(* Logix 5000 project; controller TBEN_Lx_8IOL_AOI_V0_2 vendor 1 type 14 code 176 rev 32.11; software revision 32.00; part 14 of 16 *)
(* tags used below, declared in another part *)
   TBEN_I_DATA : INT[173];   // Input Data from IO Block
   TBEN_O_DATA : INT[131];   // Output Data to IO Block
   TBEN_C_DATA : SINT[160];
   DXP1_OUT : BOOL;
   DXP3_OUT : BOOL;
   DXP5_OUT : BOOL;
   DXP7_OUT : BOOL;
   IOLDevice_PORT1 : BOOL;
   IOLDevice_PORT2 : BOOL;
   IOLDevice_PORT3 : BOOL;
   IOLDevice_PORT4 : BOOL;
   IOLDevice_PORT5 : BOOL;
   IOLDevice_PORT6 : BOOL;
   IOLDevice_PORT7 : BOOL;
   IOLDevice_PORT8 : BOOL;
   IOL0_DI : BOOL;
   DXP1_IN : BOOL;
   IOL2_DI : BOOL;
   DXP3_IN : BOOL;
   IOL4_DI : BOOL;
   DXP5_IN : BOOL;
   IOL6_DI : BOOL;
   DXP7_IN : BOOL;
   IOL8_DI : BOOL;
   IOL10_DI : BOOL;
   IOL12_DI : BOOL;
   IOL14_DI : BOOL;
   PORT1_Mode_IOL_or_DI : BOOL;   // 0: IO-LINK without validation 1: Port is set to DI (Power Cycle or Module Inhibit cycle require)
   PORT2_Mode_IOL_or_DI : BOOL;   // 0: IO-LINK without validation 1: Port is set to DI (Power Cycle or Module Inhibit cycle require)
   PORT3_Mode_IOL_or_DI : BOOL;   // 0: IO-LINK without validation 1: Port is set to DI (Power Cycle or Module Inhibit cycle require)
   PORT4_Mode_IOL_or_DI : BOOL;   // 0: IO-LINK without validation 1: Port is set to DI (Power Cycle or Module Inhibit cycle require)
   PORT5_Mode_IOL_or_DI : BOOL;   // 0: IO-LINK without validation 1: Port is set to DI (Power Cycle or Module Inhibit cycle require)
   PORT6_Mode_IOL_or_DI : BOOL;   // 0: IO-LINK without validation 1: Port is set to DI (Power Cycle or Module Inhibit cycle require)
   PORT7_Mode_IOL_or_DI : BOOL;   // 0: IO-LINK without validation 1: Port is set to DI (Power Cycle or Module Inhibit cycle require)
   PORT8_Mode_IOL_or_DI : BOOL;   // 0: IO-LINK without validation 1: Port is set to DI (Power Cycle or Module Inhibit cycle require)
   DisableOutput_DXP1 : BOOL;
   DisableOutput_DXP3 : BOOL;
   DisableOutput_DXP5 : BOOL;
   DisableOutput_DXP7 : BOOL;
   IOLReadActive : BOOL;
   IOLWriteActive : BOOL;
   IOL_READ_Request : BOOL;
   IOL_WRITE_Request : BOOL;
(* TBEN_Lx_8IOL_AOI, continued *)

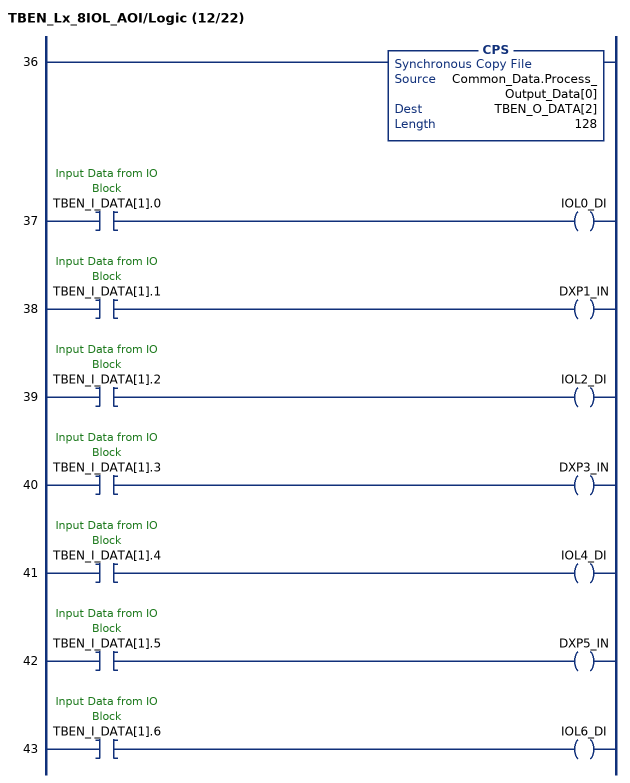
   36: CPS(Common_Data.Process_Output_Data[0],TBEN_O_DATA[2],128);
   37: XIC(TBEN_I_DATA[1].0)OTE(IOL0_DI);
   38: XIC(TBEN_I_DATA[1].1)OTE(DXP1_IN);
   39: XIC(TBEN_I_DATA[1].2)OTE(IOL2_DI);
   40: XIC(TBEN_I_DATA[1].3)OTE(DXP3_IN);
   41: XIC(TBEN_I_DATA[1].4)OTE(IOL4_DI);
   42: XIC(TBEN_I_DATA[1].5)OTE(DXP5_IN);
   43: XIC(TBEN_I_DATA[1].6)OTE(IOL6_DI);
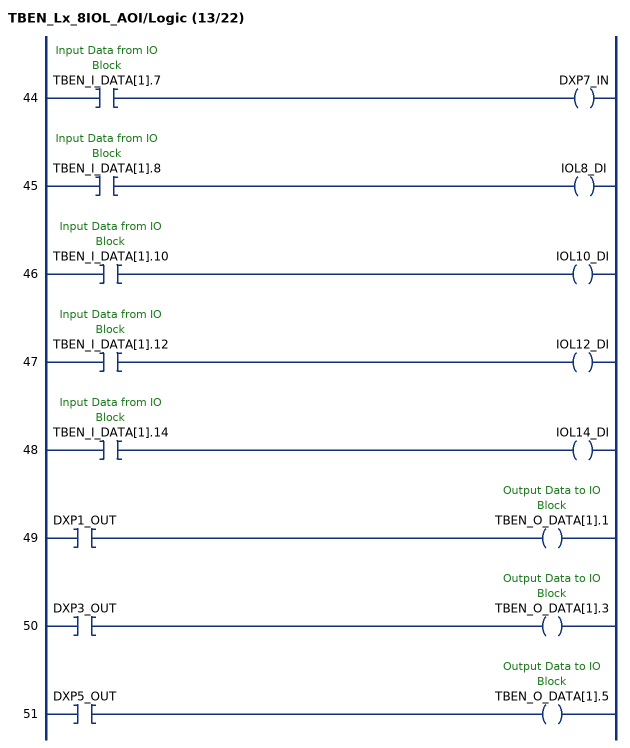
   44: XIC(TBEN_I_DATA[1].7)OTE(DXP7_IN);
   45: XIC(TBEN_I_DATA[1].8)OTE(IOL8_DI);
   46: XIC(TBEN_I_DATA[1].10)OTE(IOL10_DI);
   47: XIC(TBEN_I_DATA[1].12)OTE(IOL12_DI);
   48: XIC(TBEN_I_DATA[1].14)OTE(IOL14_DI);
   49: XIC(DXP1_OUT)OTE(TBEN_O_DATA[1].1);
   50: XIC(DXP3_OUT)OTE(TBEN_O_DATA[1].3);
   51: XIC(DXP5_OUT)OTE(TBEN_O_DATA[1].5);
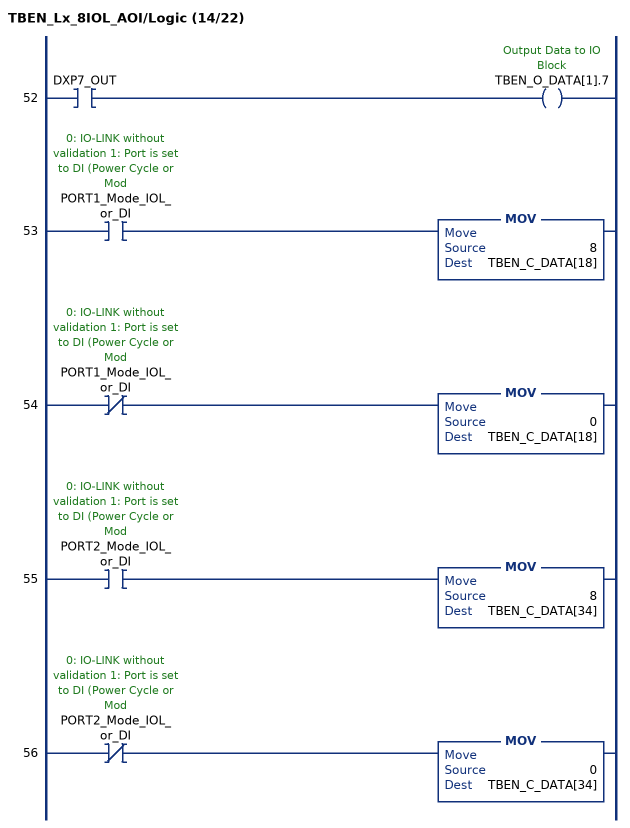
   52: XIC(DXP7_OUT)OTE(TBEN_O_DATA[1].7);
   53: XIC(PORT1_Mode_IOL_or_DI)MOV(8,TBEN_C_DATA[18]);
   54: XIO(PORT1_Mode_IOL_or_DI)MOV(0,TBEN_C_DATA[18]);
   55: XIC(PORT2_Mode_IOL_or_DI)MOV(8,TBEN_C_DATA[34]);
   56: XIO(PORT2_Mode_IOL_or_DI)MOV(0,TBEN_C_DATA[34]);
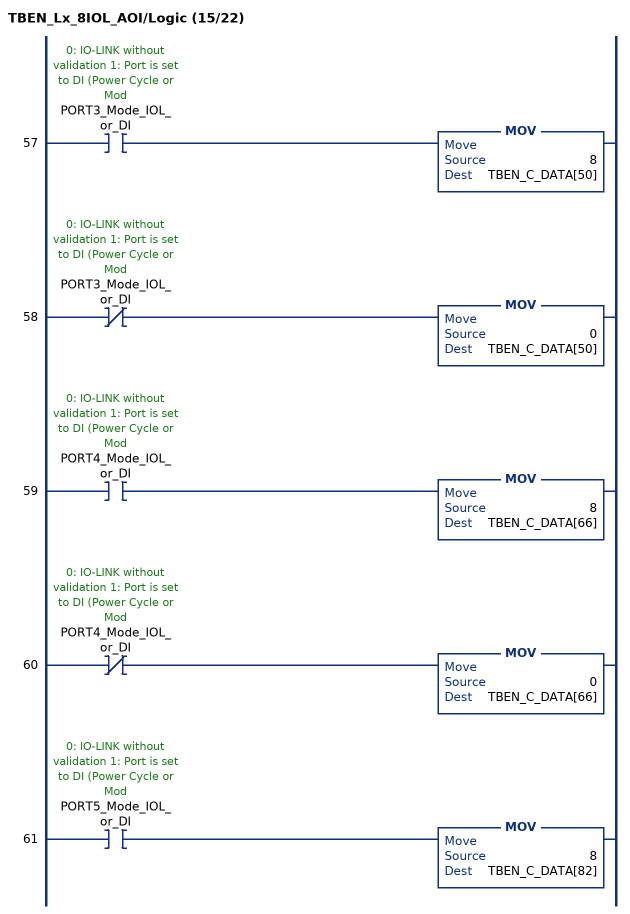
   57: XIC(PORT3_Mode_IOL_or_DI)MOV(8,TBEN_C_DATA[50]);
   58: XIO(PORT3_Mode_IOL_or_DI)MOV(0,TBEN_C_DATA[50]);
   59: XIC(PORT4_Mode_IOL_or_DI)MOV(8,TBEN_C_DATA[66]);
   60: XIO(PORT4_Mode_IOL_or_DI)MOV(0,TBEN_C_DATA[66]);
   61: XIC(PORT5_Mode_IOL_or_DI)MOV(8,TBEN_C_DATA[82]);
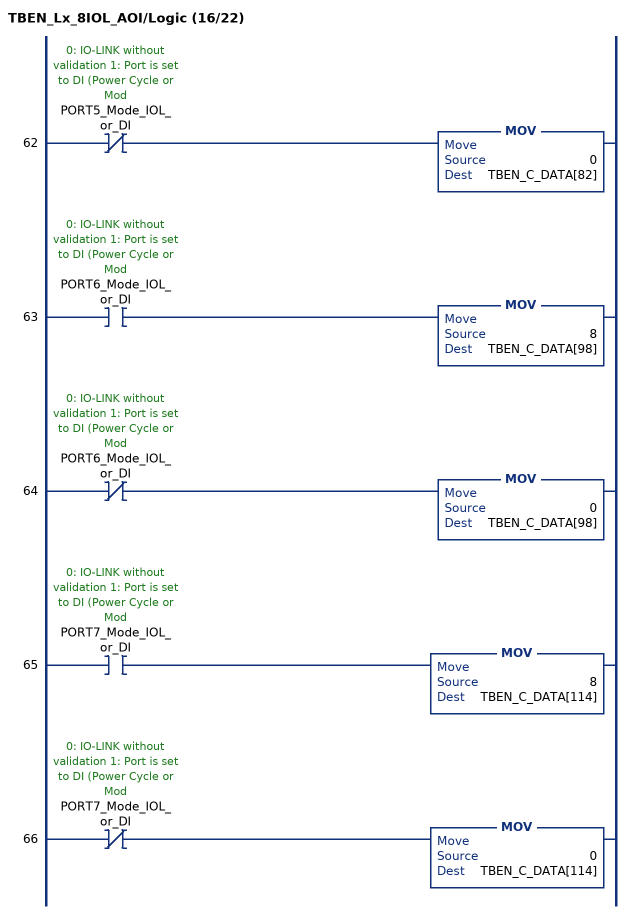
   62: XIO(PORT5_Mode_IOL_or_DI)MOV(0,TBEN_C_DATA[82]);
   63: XIC(PORT6_Mode_IOL_or_DI)MOV(8,TBEN_C_DATA[98]);
   64: XIO(PORT6_Mode_IOL_or_DI)MOV(0,TBEN_C_DATA[98]);
   65: XIC(PORT7_Mode_IOL_or_DI)MOV(8,TBEN_C_DATA[114]);
   66: XIO(PORT7_Mode_IOL_or_DI)MOV(0,TBEN_C_DATA[114]);
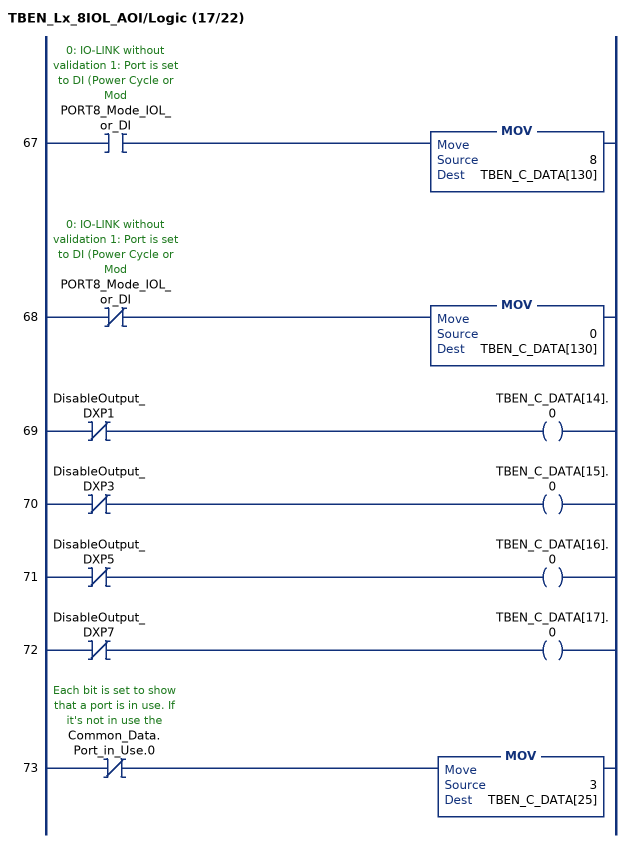
   67: XIC(PORT8_Mode_IOL_or_DI)MOV(8,TBEN_C_DATA[130]);
   68: XIO(PORT8_Mode_IOL_or_DI)MOV(0,TBEN_C_DATA[130]);
   69: XIO(DisableOutput_DXP1)OTE(TBEN_C_DATA[14].0);
   70: XIO(DisableOutput_DXP3)OTE(TBEN_C_DATA[15].0);
   71: XIO(DisableOutput_DXP5)OTE(TBEN_C_DATA[16].0);
   72: XIO(DisableOutput_DXP7)OTE(TBEN_C_DATA[17].0);
   73: XIO(Common_Data.Port_in_Use.0)MOV(3,TBEN_C_DATA[25]);
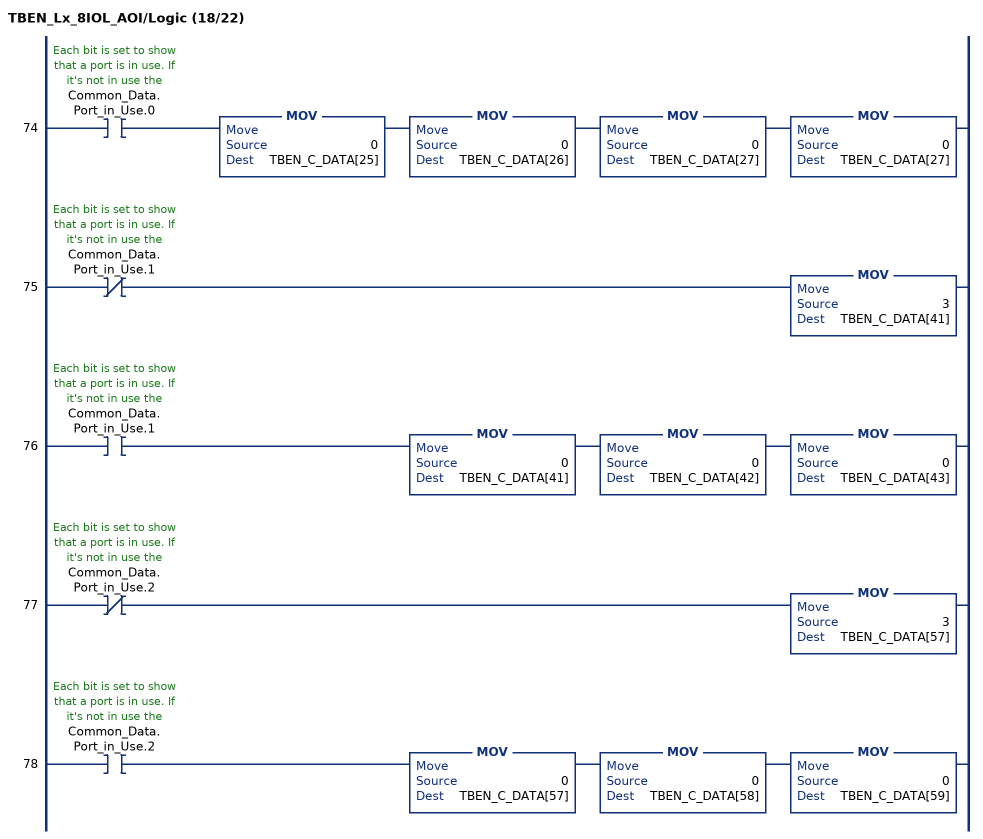
   74: XIC(Common_Data.Port_in_Use.0)MOV(0,TBEN_C_DATA[25])MOV(0,TBEN_C_DATA[26])MOV(0,TBEN_C_DATA[27])MOV(0,TBEN_C_DATA[27]);
   75: XIO(Common_Data.Port_in_Use.1)MOV(3,TBEN_C_DATA[41]);
   76: XIC(Common_Data.Port_in_Use.1)MOV(0,TBEN_C_DATA[41])MOV(0,TBEN_C_DATA[42])MOV(0,TBEN_C_DATA[43]);
   77: XIO(Common_Data.Port_in_Use.2)MOV(3,TBEN_C_DATA[57]);
   78: XIC(Common_Data.Port_in_Use.2)MOV(0,TBEN_C_DATA[57])MOV(0,TBEN_C_DATA[58])MOV(0,TBEN_C_DATA[59]);
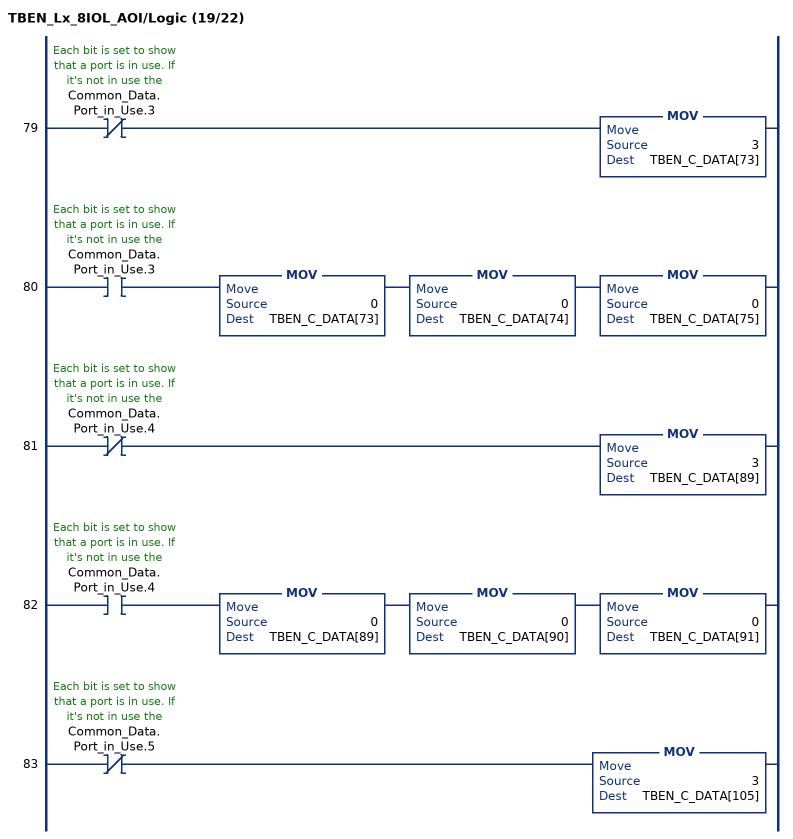
   79: XIO(Common_Data.Port_in_Use.3)MOV(3,TBEN_C_DATA[73]);
   80: XIC(Common_Data.Port_in_Use.3)MOV(0,TBEN_C_DATA[73])MOV(0,TBEN_C_DATA[74])MOV(0,TBEN_C_DATA[75]);
   81: XIO(Common_Data.Port_in_Use.4)MOV(3,TBEN_C_DATA[89]);
   82: XIC(Common_Data.Port_in_Use.4)MOV(0,TBEN_C_DATA[89])MOV(0,TBEN_C_DATA[90])MOV(0,TBEN_C_DATA[91]);
   83: XIO(Common_Data.Port_in_Use.5)MOV(3,TBEN_C_DATA[105]);
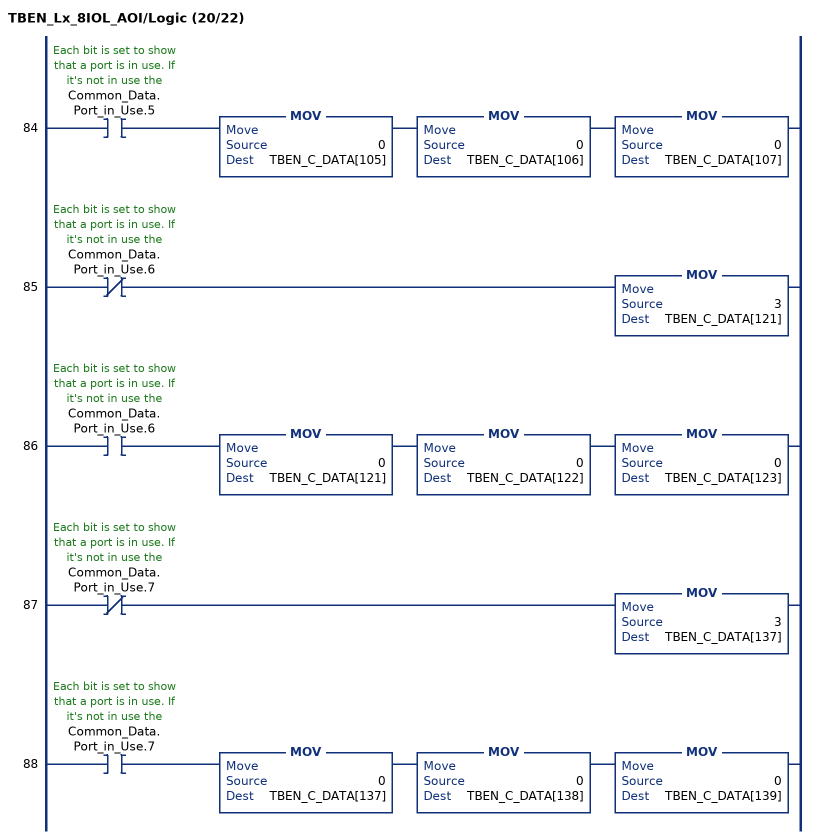
   84: XIC(Common_Data.Port_in_Use.5)MOV(0,TBEN_C_DATA[105])MOV(0,TBEN_C_DATA[106])MOV(0,TBEN_C_DATA[107]);
   85: XIO(Common_Data.Port_in_Use.6)MOV(3,TBEN_C_DATA[121]);
   86: XIC(Common_Data.Port_in_Use.6)MOV(0,TBEN_C_DATA[121])MOV(0,TBEN_C_DATA[122])MOV(0,TBEN_C_DATA[123]);
   87: XIO(Common_Data.Port_in_Use.7)MOV(3,TBEN_C_DATA[137]);
   88: XIC(Common_Data.Port_in_Use.7)MOV(0,TBEN_C_DATA[137])MOV(0,TBEN_C_DATA[138])MOV(0,TBEN_C_DATA[139]);
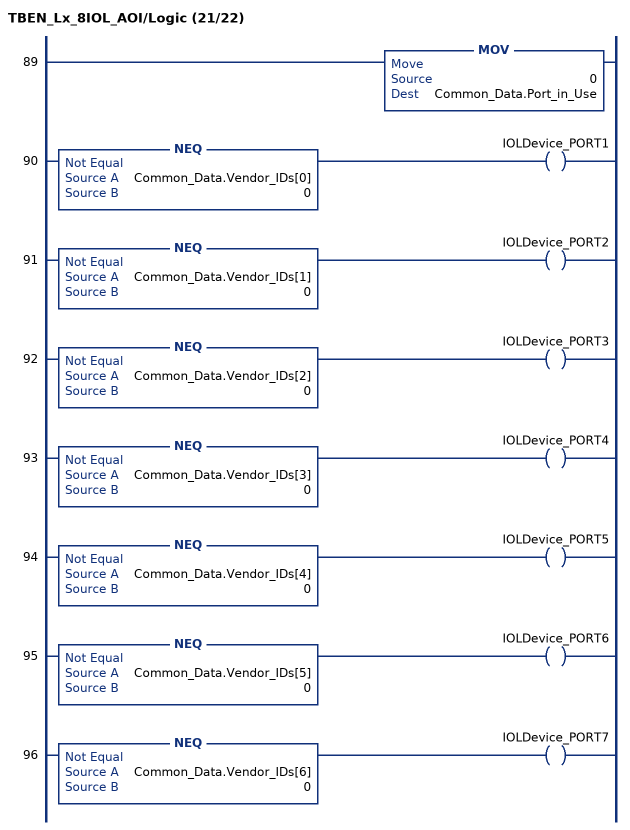
   89: MOV(0,Common_Data.Port_in_Use);
   90: NEQ(Common_Data.Vendor_IDs[0],0)OTE(IOLDevice_PORT1);
   91: NEQ(Common_Data.Vendor_IDs[1],0)OTE(IOLDevice_PORT2);
   92: NEQ(Common_Data.Vendor_IDs[2],0)OTE(IOLDevice_PORT3);
   93: NEQ(Common_Data.Vendor_IDs[3],0)OTE(IOLDevice_PORT4);
   94: NEQ(Common_Data.Vendor_IDs[4],0)OTE(IOLDevice_PORT5);
   95: NEQ(Common_Data.Vendor_IDs[5],0)OTE(IOLDevice_PORT6);
   96: NEQ(Common_Data.Vendor_IDs[6],0)OTE(IOLDevice_PORT7);
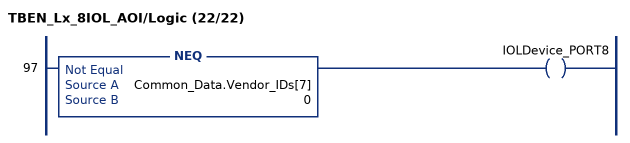
   97: NEQ(Common_Data.Vendor_IDs[7],0)OTE(IOLDevice_PORT8);
END_ROUTINE

ROUTINE Prescan   (* ladder *)
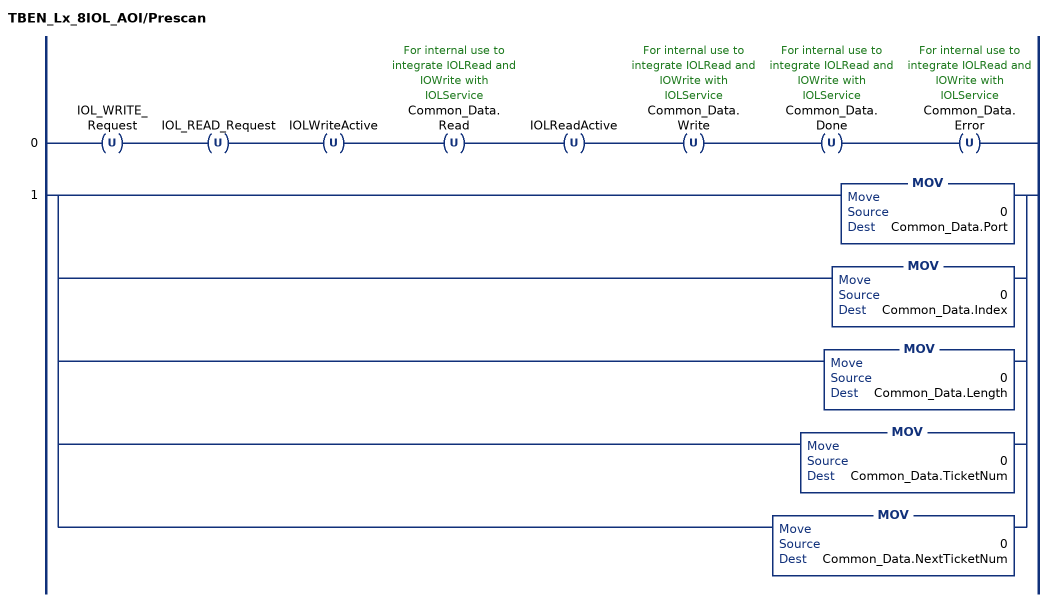
   0: OTU(IOL_WRITE_Request)OTU(IOL_READ_Request)OTU(IOLWriteActive)OTU(Common_Data.Read)OTU(IOLReadActive)OTU(Common_Data.Write)OTU(Common_Data.Done)OTU(Common_Data.Error);
   1: [MOV(0,Common_Data.Port) ,MOV(0,Common_Data.Index) ,MOV(0,Common_Data.Length) ,MOV(0,Common_Data.TicketNum) ,MOV(0,Common_Data.NextTicketNum) ];
END_ROUTINE
END_ADD_ON_INSTRUCTION

ADD_ON_INSTRUCTION Universal_Device_Info   (* revision 1.0, ExecutePrescan *)
VAR_INPUT
   Port : INT; {required}
END_VAR
VAR_IN_OUT
   Common_Data : Turck_IOLink_Common_Data; {required}
END_VAR
VAR_INPUT
   Write_Application_Specific_Tag : BOOL;
END_VAR
VAR_IN_OUT
   Universal_IOLink_Info : Universal_IOLink_Info; {required}
END_VAR
VAR
   StartupDone : BOOL; {access None}
   Done : DINT; {access None}
   Error : DINT; {access None}
   Active : DINT; {access None}
   Pending : DINT; {access None}
   Pending_or_Active : DINT; {access None}
   StartupCount : DINT; {access None}
   MyTicketNum : DINT[32]; {access None}
   Read_ONS : DINT; {access None}
   ReadRequest : DINT; {access None}
   Read : DINT; {access None}
   DoneCount : DINT; {access None}
   Status : DINT; {access None}
   ErrorCount : DINT; {access None}
   Prev_Vendor_ID : INT; {access None}
   Update_Data : BOOL; {access None}
   Reset : BOOL; {access None}
   Write_ONS : DINT; {access None}
   WriteRequest : DINT; {access None}
END_VAR

ROUTINE Logic   (* ladder *)
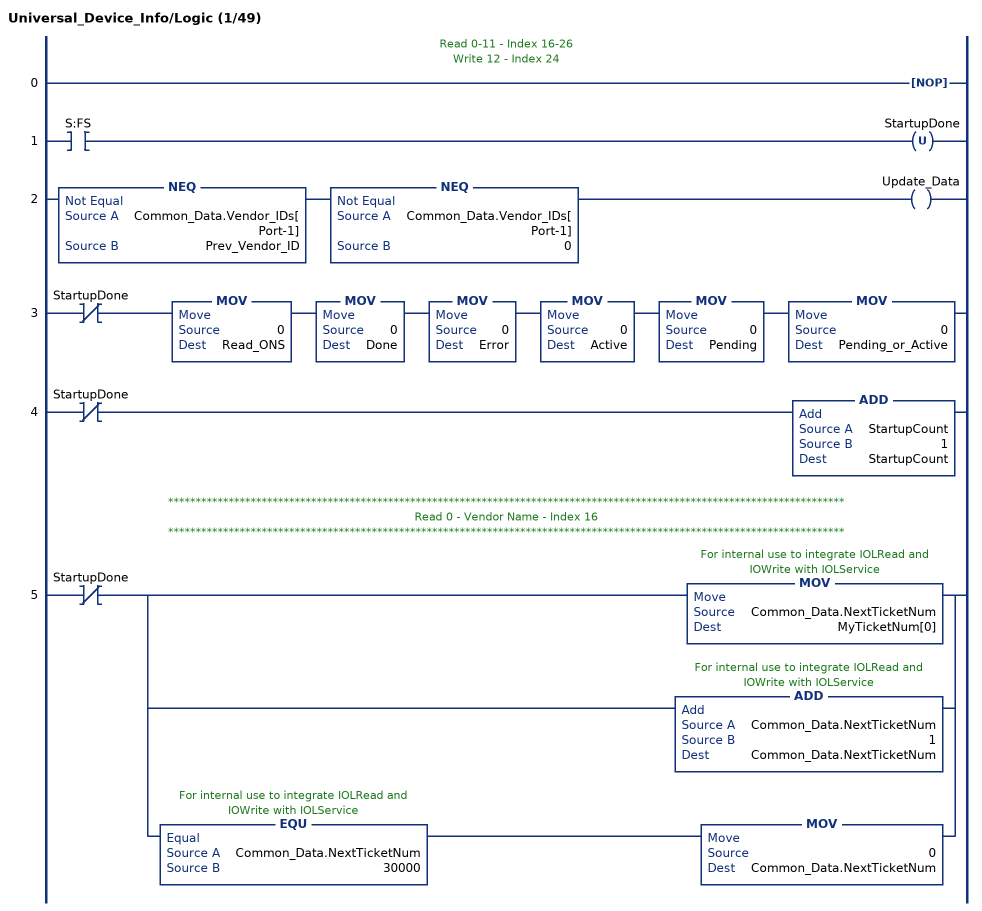
   // Read 0-11 - Index 16-26
   // Write 12 - Index 24
   0: NOP();
   1: XIC(S:FS)OTU(StartupDone);
   2: NEQ(Common_Data.Vendor_IDs[Port-1],Prev_Vendor_ID)NEQ(Common_Data.Vendor_IDs[Port-1],0)OTE(Update_Data);
   3: XIO(StartupDone)MOV(0,Read_ONS)MOV(0,Done)MOV(0,Error)MOV(0,Active)MOV(0,Pending)MOV(0,Pending_or_Active);
   4: XIO(StartupDone)ADD(StartupCount,1,StartupCount);
   // ***************************************************************************************************************************
   // Read 0 - Vendor Name - Index 16
   // ***************************************************************************************************************************
   5: XIO(StartupDone)[MOV(Common_Data.NextTicketNum,MyTicketNum[0]) ,ADD(Common_Data.NextTicketNum,1,Common_Data.NextTicketNum) ,EQU(Common_Data.NextTicketNum,30000) MOV(0,Common_Data.NextTicketNum) ];
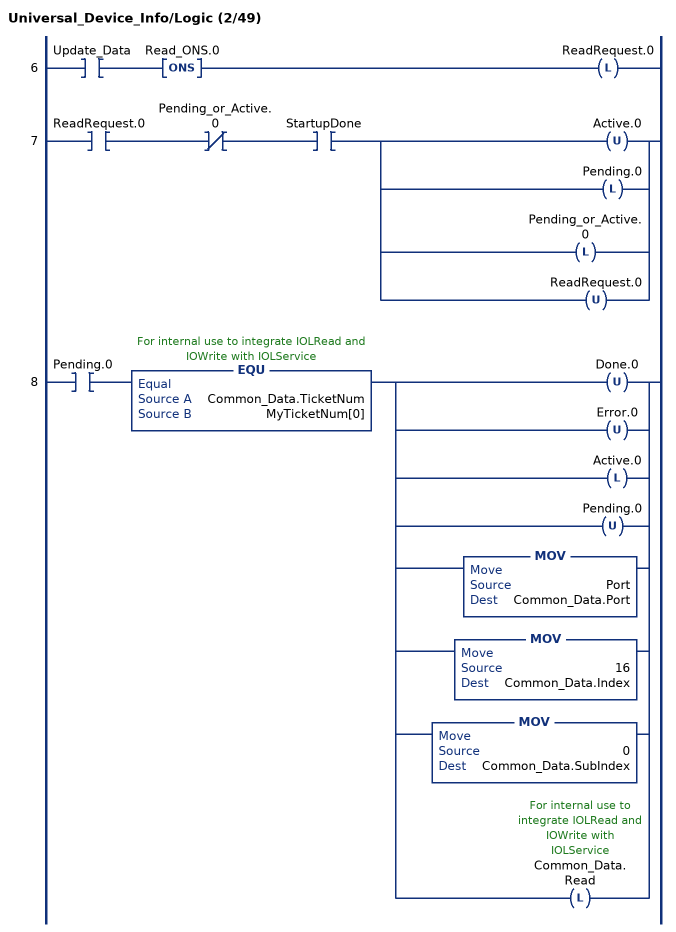
   6: XIC(Update_Data)ONS(Read_ONS.0)OTL(ReadRequest.0);
   7: XIC(ReadRequest.0)XIO(Pending_or_Active.0)XIC(StartupDone)[OTU(Active.0) ,OTL(Pending.0) ,OTL(Pending_or_Active.0) ,OTU(ReadRequest.0) ];
   8: XIC(Pending.0)EQU(Common_Data.TicketNum,MyTicketNum[0])[OTU(Done.0) ,OTU(Error.0) ,OTL(Active.0) ,OTU(Pending.0) ,MOV(Port,Common_Data.Port) ,MOV(16,Common_Data.Index) ,MOV(0,Common_Data.SubIndex) ,OTL(Common_Data.Read) ];
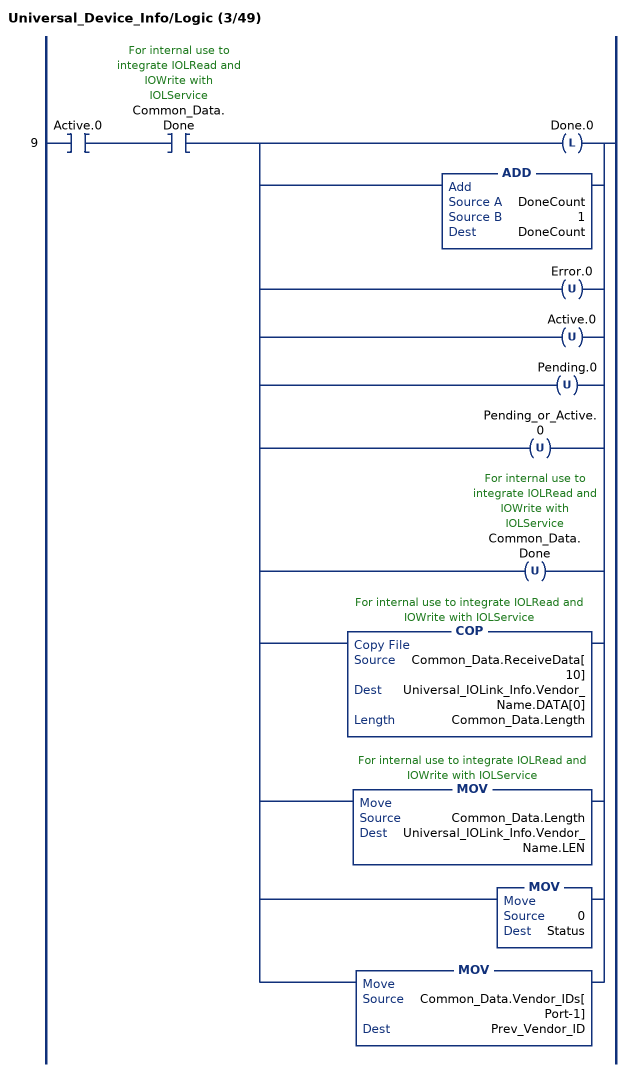
   9: XIC(Active.0)XIC(Common_Data.Done)[OTL(Done.0) ,ADD(DoneCount,1,DoneCount) ,OTU(Error.0) ,OTU(Active.0) ,OTU(Pending.0) ,OTU(Pending_or_Active.0) ,OTU(Common_Data.Done) ,COP(Common_Data.ReceiveData[10],Universal_IOLink_Info.Vendor_Name.DATA[0],Common_Data.Length) ,MOV(Common_Data.Length,Universal_IOLink_Info.Vendor_Name.LEN) ,MOV(0,Status) ,MOV(Common_Data.Vendor_IDs[Port-1],Prev_Vendor_ID) ];
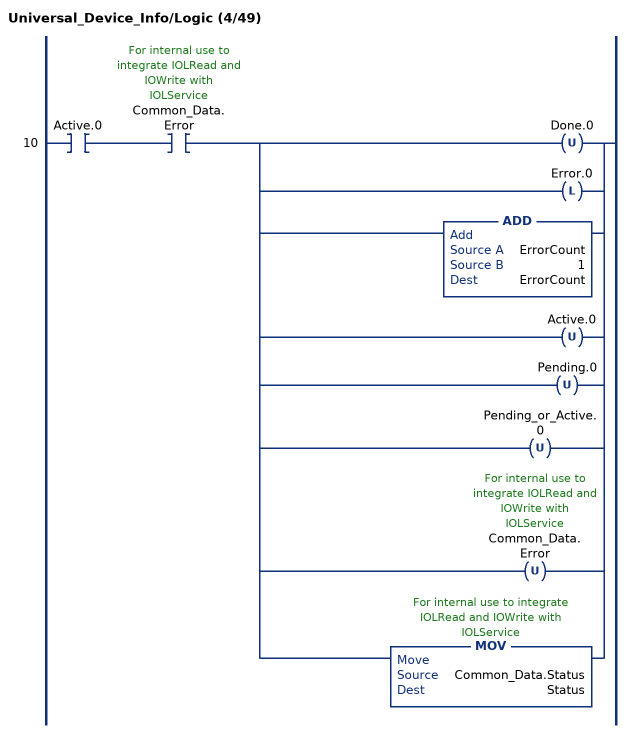
   10: XIC(Active.0)XIC(Common_Data.Error)[OTU(Done.0) ,OTL(Error.0) ,ADD(ErrorCount,1,ErrorCount) ,OTU(Active.0) ,OTU(Pending.0) ,OTU(Pending_or_Active.0) ,OTU(Common_Data.Error) ,MOV(Common_Data.Status,Status) ];
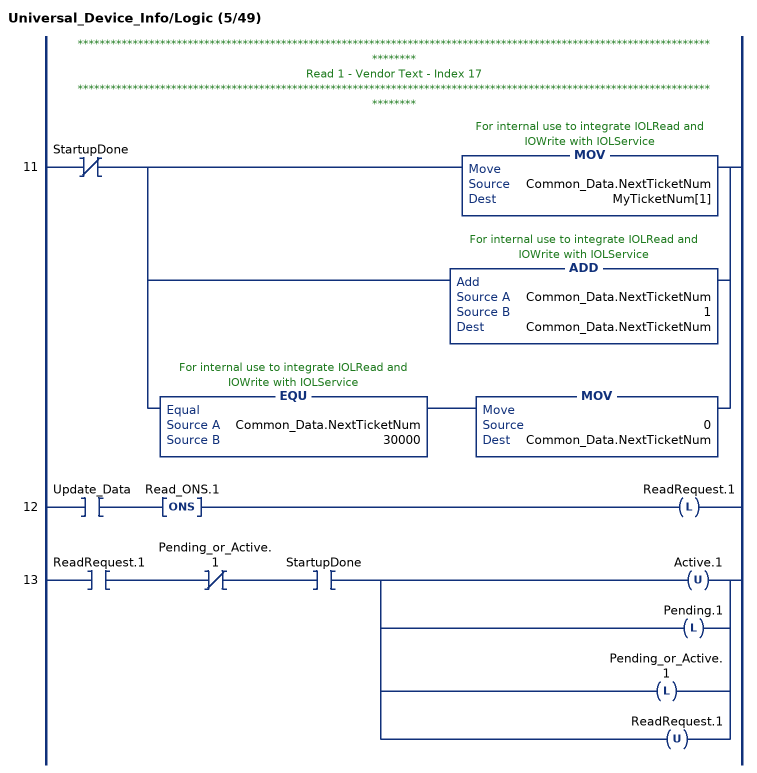
   // ***************************************************************************************************************************
   // Read 1 - Vendor Text - Index 17
   // ***************************************************************************************************************************
   11: XIO(StartupDone)[MOV(Common_Data.NextTicketNum,MyTicketNum[1]) ,ADD(Common_Data.NextTicketNum,1,Common_Data.NextTicketNum) ,EQU(Common_Data.NextTicketNum,30000) MOV(0,Common_Data.NextTicketNum) ];
   12: XIC(Update_Data)ONS(Read_ONS.1)OTL(ReadRequest.1);
   13: XIC(ReadRequest.1)XIO(Pending_or_Active.1)XIC(StartupDone)[OTU(Active.1) ,OTL(Pending.1) ,OTL(Pending_or_Active.1) ,OTU(ReadRequest.1) ];
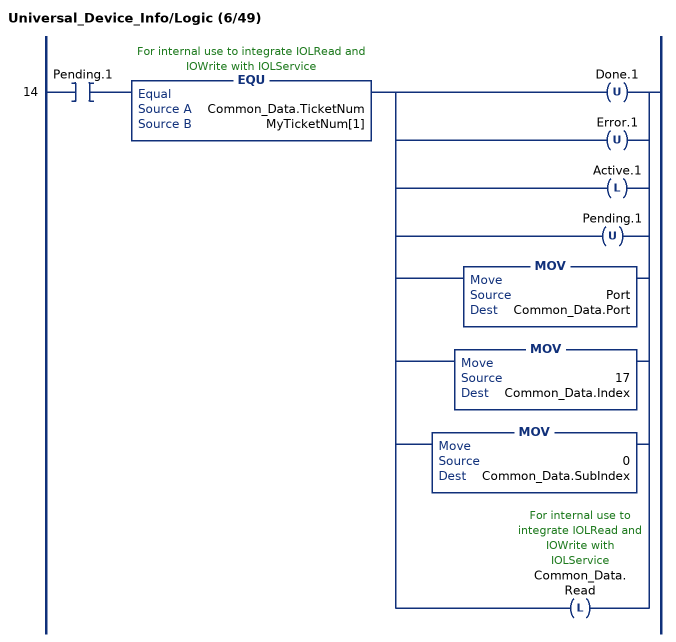
   14: XIC(Pending.1)EQU(Common_Data.TicketNum,MyTicketNum[1])[OTU(Done.1) ,OTU(Error.1) ,OTL(Active.1) ,OTU(Pending.1) ,MOV(Port,Common_Data.Port) ,MOV(17,Common_Data.Index) ,MOV(0,Common_Data.SubIndex) ,OTL(Common_Data.Read) ];
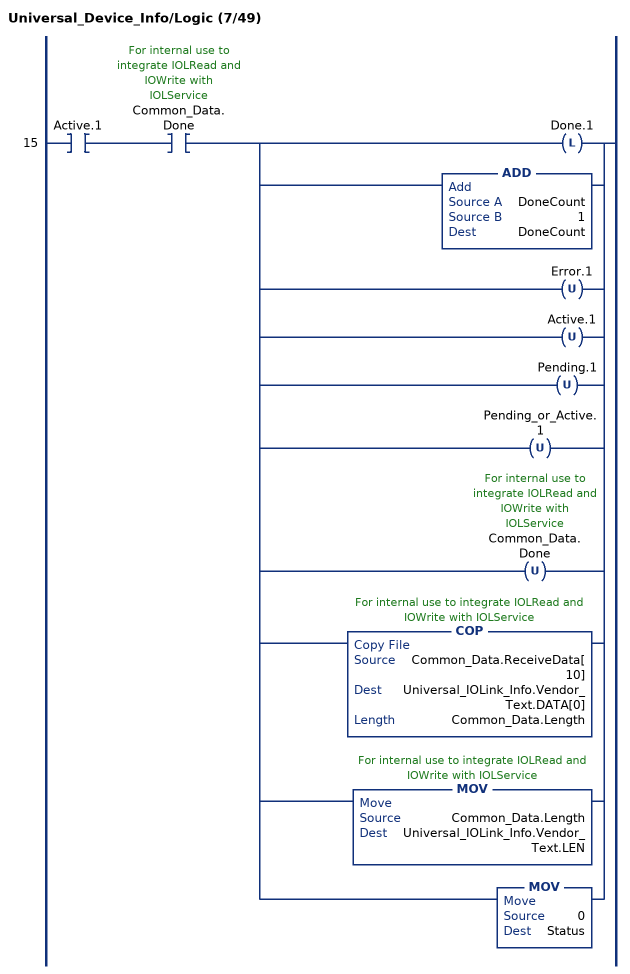
   15: XIC(Active.1)XIC(Common_Data.Done)[OTL(Done.1) ,ADD(DoneCount,1,DoneCount) ,OTU(Error.1) ,OTU(Active.1) ,OTU(Pending.1) ,OTU(Pending_or_Active.1) ,OTU(Common_Data.Done) ,COP(Common_Data.ReceiveData[10],Universal_IOLink_Info.Vendor_Text.DATA[0],Common_Data.Length) ,MOV(Common_Data.Length,Universal_IOLink_Info.Vendor_Text.LEN) ,MOV(0,Status) ];
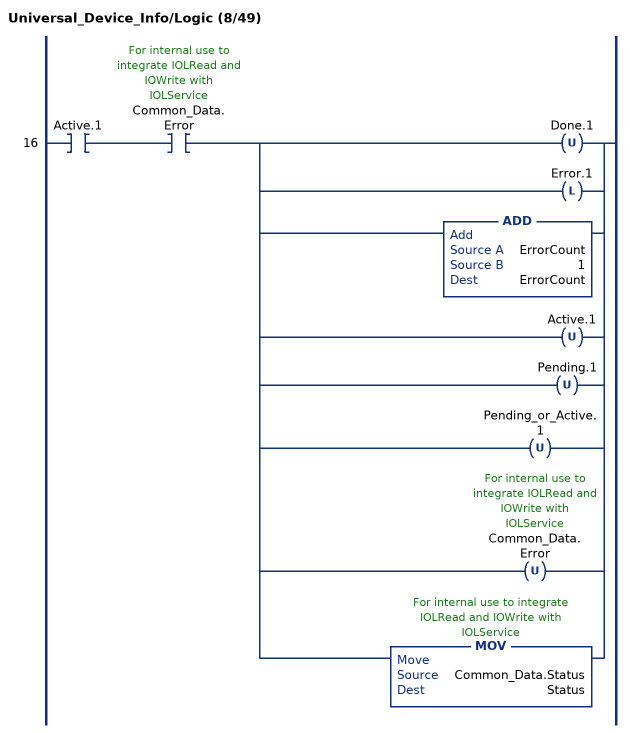
   16: XIC(Active.1)XIC(Common_Data.Error)[OTU(Done.1) ,OTL(Error.1) ,ADD(ErrorCount,1,ErrorCount) ,OTU(Active.1) ,OTU(Pending.1) ,OTU(Pending_or_Active.1) ,OTU(Common_Data.Error) ,MOV(Common_Data.Status,Status) ];
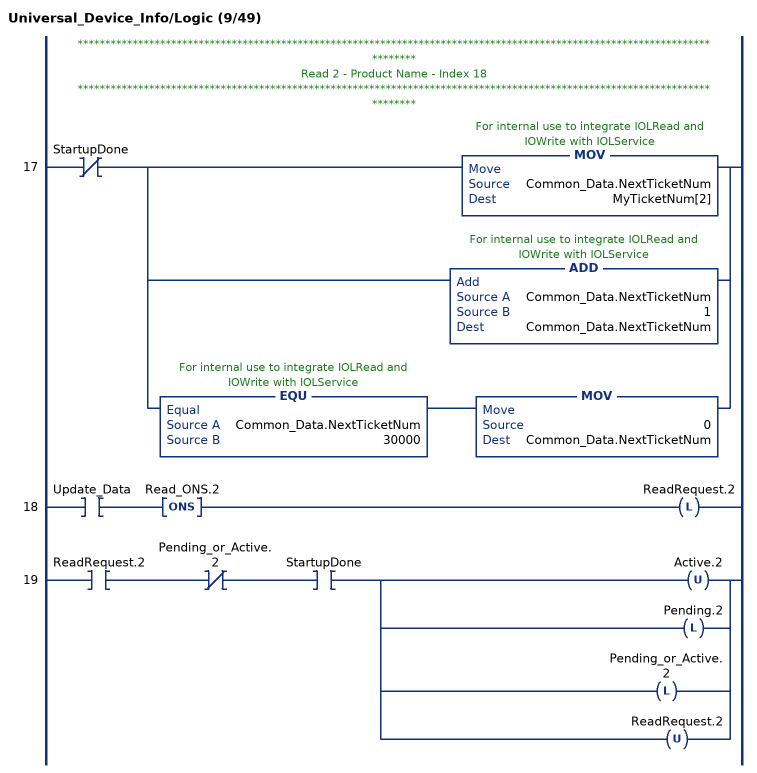
   // ***************************************************************************************************************************
   // Read 2 - Product Name - Index 18
   // ***************************************************************************************************************************
   17: XIO(StartupDone)[MOV(Common_Data.NextTicketNum,MyTicketNum[2]) ,ADD(Common_Data.NextTicketNum,1,Common_Data.NextTicketNum) ,EQU(Common_Data.NextTicketNum,30000) MOV(0,Common_Data.NextTicketNum) ];
   18: XIC(Update_Data)ONS(Read_ONS.2)OTL(ReadRequest.2);
   19: XIC(ReadRequest.2)XIO(Pending_or_Active.2)XIC(StartupDone)[OTU(Active.2) ,OTL(Pending.2) ,OTL(Pending_or_Active.2) ,OTU(ReadRequest.2) ];
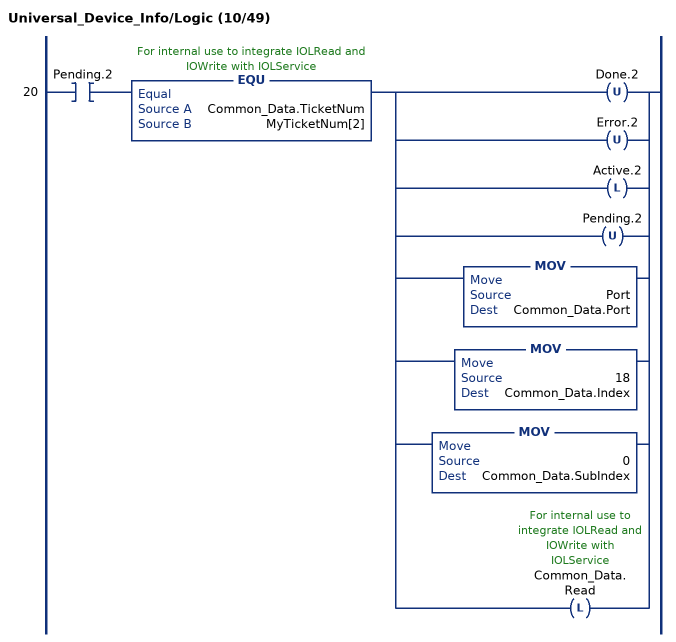
   20: XIC(Pending.2)EQU(Common_Data.TicketNum,MyTicketNum[2])[OTU(Done.2) ,OTU(Error.2) ,OTL(Active.2) ,OTU(Pending.2) ,MOV(Port,Common_Data.Port) ,MOV(18,Common_Data.Index) ,MOV(0,Common_Data.SubIndex) ,OTL(Common_Data.Read) ];
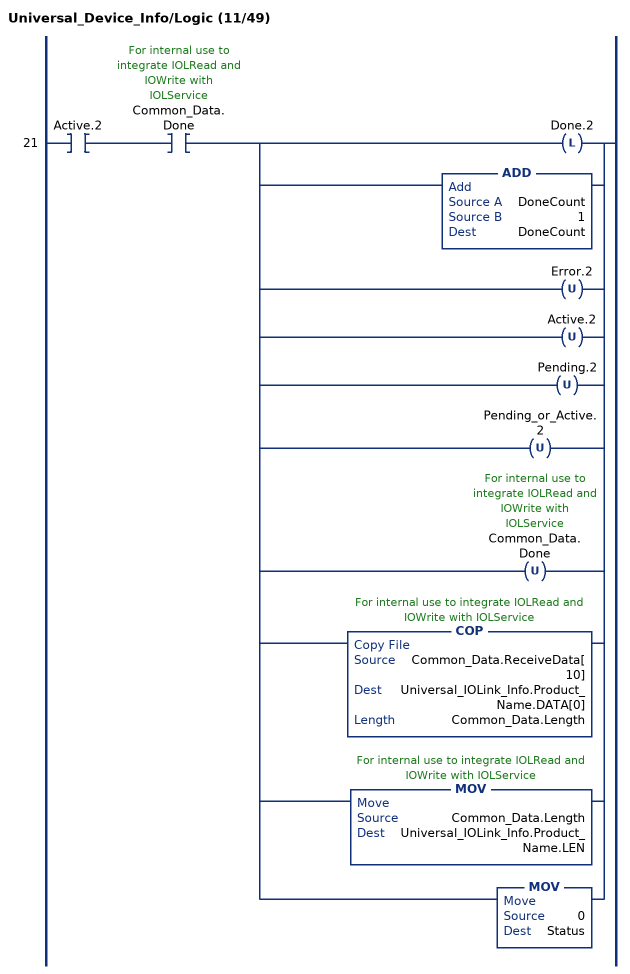
   21: XIC(Active.2)XIC(Common_Data.Done)[OTL(Done.2) ,ADD(DoneCount,1,DoneCount) ,OTU(Error.2) ,OTU(Active.2) ,OTU(Pending.2) ,OTU(Pending_or_Active.2) ,OTU(Common_Data.Done) ,COP(Common_Data.ReceiveData[10],Universal_IOLink_Info.Product_Name.DATA[0],Common_Data.Length) ,MOV(Common_Data.Length,Universal_IOLink_Info.Product_Name.LEN) ,MOV(0,Status) ];
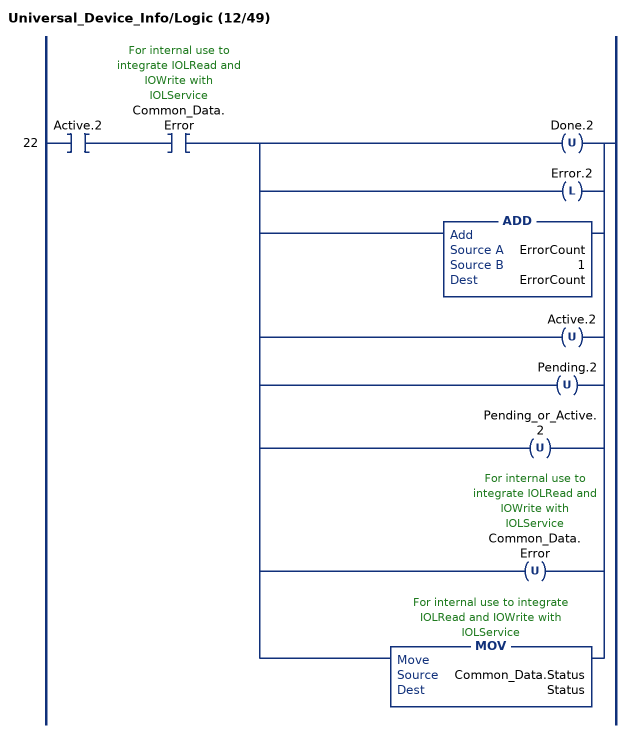
   22: XIC(Active.2)XIC(Common_Data.Error)[OTU(Done.2) ,OTL(Error.2) ,ADD(ErrorCount,1,ErrorCount) ,OTU(Active.2) ,OTU(Pending.2) ,OTU(Pending_or_Active.2) ,OTU(Common_Data.Error) ,MOV(Common_Data.Status,Status) ];
